// TIA Portal V19 export
FUNCTION "OutputHandler3" : Void   // FC55, STL
TITLE = OutputHandler3
{ S7_Optimized_Access := 'TRUE' }
// IO-Link Items i.e Valves and process instruments in "IO-Link Devices"FB10
// stored: AutoNumber false
   VAR_TEMP
      V0945_closed : Bool;
      M0941_NotRunning : Bool;
   END_VAR
BEGIN

NETWORK
TITLE = # V0945_closed
      A     "PG_Devices".V0945_SV2;
      AN    "PG_Devices".V0945_Closed;
      O     "PG_Devices".V0945_Closed;
      =     #V0945_closed;

NETWORK
TITLE = V0945 - Bardiarni
// CALL  "Item_Control"
//        DATAWORD  :=DBW150
//        RESET_IRES:=#V0945_closed
//        SET_INPUT :="PG_Devices".V0945_Open
//        _TYPE     :=2
//        MAX_TIME  :=3
//        OUTPUT    :="PG_Devices".V0945_SV1
      CALL  "Item_Control"
      ( "type"      := 1,
        maxTime     := 5,
        itemInfo    := "ItemInfoScada".Items[76],
        itemTimer   := "ItemTimerwork".V0945,
        itemStatus  := "ItemStatus".V0945,
        itemCommand := "ItemCommand".V0945,
        resetInput  := "PG_Devices".V0945_Closed,
        setInput    := "PG_Devices".V0945_Open,
        output      := "PG_Devices".V0945_SV1
      );


NETWORK
TITLE = M0940
// This aligns with network 12 in "ControlAutobit3" FC54
      CALL  "VSD Item Control", "M0940 G120_DI"
      ( tripped     := "PG_Devices".DI_100_010_X01_4,
        iso_On      := "PG_Devices".M0940_Iso,
        maxTime     := 10,
        rpm_Sp      := "PID_Loops_DB".RPM,
        hwID        := "9~M0940~M09_40_VSD",
        output      := ,
        ItemInfo    := "ItemInfoScada".Items[77],
        ItemTimer   := "ItemTimerwork".M0940,
        ItemStatus  := "ItemStatus".M0940,
        ItemCommand := "ItemCommand".M0940
      );






NETWORK
TITLE = M0940 Parameter Read
      CALL  SinaPara, "SinaPara_IDB"
      ( Start      := "readwrite_hmi_interface".start,
        ReadWrite  := 0,
        ParaNo     := 945,
        AxisNo     := 1,
        hardwareId := "9~M0940~M09_40_VSD",
        Ready      := ,
        Busy       := "readwrite_hmi_interface".busy,
        Done       := "readwrite_hmi_interface".done,
        Error      := "readwrite_hmi_interface".error,
        ErrorId    := "readwrite_hmi_interface".errorID,
        DiagId     := ,
        Parameter  := "answer_from_drive_read".FaultBuffer
      );



NETWORK
TITLE = M0941
// This aligns with network 19 in "ControlAutobit3" FC54
      L     "Tag_12":P;
      T     "Tag_12";

// Isolator HMI Indication
      AN    "PG_Devices".M0941_Iso;
      =     "ItemInfoScada".Items[84].IsolatedInd;

      AN    "I553.0";
      =     #M0941_NotRunning;

      CALL  "Item_Control"
      ( "type"      := 3,  // 0=NO-FB, 1=SET-FB, 2=RES-FB, 3=S/R-FB
        maxTime     := 10,  // Max feed-back MAX_TIME
        itemInfo    := "ItemInfoScada".Items[84],  //M0941
        itemTimer   := "ItemTimerwork".M0941,
        itemStatus  := "ItemStatus".M0941,
        itemCommand := "ItemCommand".M0941,
        resetInput  := #M0941_NotRunning,  // Input for de-energised feed-back
        setInput    := "I553.0",  // Input for energised feed-back
        output      := "Tag_81"  // Output
      );

      L     "Tag_29";
      T     "Tag_29":P;
      T     "Tag_14":P;


END_FUNCTION
